FUNCTION_BLOCK OPTIMIZER
  {SET_ATTRIBUTE(OpcUa, SERVICE)}
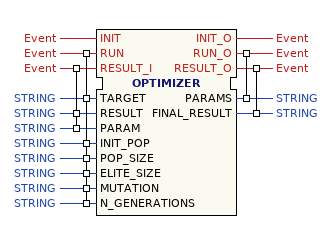
  EVENT_INPUT
    INIT;
    RUN WITH TARGET, INIT_POP, POP_SIZE, ELITE_SIZE, MUTATION, N_GENERATIONS;
    RESULT_I WITH RESULT, PARAM;
  END_EVENT
  EVENT_OUTPUT
    INIT_O;
    RUN_O WITH PARAMS;
    RESULT_O WITH FINAL_RESULT;
  END_EVENT
  VAR_INPUT
    TARGET : STRING; {SET_ATTRIBUTE(OpcUa, Constant)}
    RESULT : STRING; {SET_ATTRIBUTE(OpcUa, Variable)}
    PARAM : STRING; {SET_ATTRIBUTE(OpcUa, Variable)}
    INIT_POP : STRING; {SET_ATTRIBUTE(OpcUa, Constant)}
    POP_SIZE : STRING; {SET_ATTRIBUTE(OpcUa, Constant)}
    ELITE_SIZE : STRING; {SET_ATTRIBUTE(OpcUa, Constant)}
    MUTATION : STRING; {SET_ATTRIBUTE(OpcUa, Constant)}
    N_GENERATIONS : STRING; {SET_ATTRIBUTE(OpcUa, Constant)}
  END_VAR
  VAR_OUTPUT
    PARAMS : STRING; {SET_ATTRIBUTE(OpcUa, Variable)}
    FINAL_RESULT : STRING; {SET_ATTRIBUTE(OpcUa, Variable)}
  END_VAR
END_FUNCTION_BLOCK
